PROGRAM MAIN
VAR CONSTANT
	INSTANCE_NAME: STRING := 'MAIN Program';
	IGNORE_DEFINITION: BOOL := TRUE;
	IGNORE_STOP: BOOL := TRUE;
END_VAR
VAR
	// define services
	m_buttonManager: ButtonManager;
	m_errorManager: ErrorManager;
	m_services: ServiceContainer(ADR(m_errorManager));
	
	// instantiate machine behavior model
	m_container: xPPU_Container(
		m_services.PtrStateTracker, 
		m_services.PtrProcessManager, 
		ADR(m_errorManager));
	
	// INTERLOCKS - must always be False
	// (EProcessVariables.LSC_RampEndWPCount >= 3) AND ((EProcessVariables.LSC_RampStartWPCount >= 3) OR ((EProcessVariables.LSC_RampMiddleWPCount >= 3) OR (EProcessVariables.SSC_RampWPCount >= 3)))
	m_compExpr1: ComparisonExpression(EProcessVariables.LSC_RampEndWPCount, EComparisonType.greater_eq, EDataType.numeric, FALSE, 3, '', TRUE);
	m_compExpr3: ComparisonExpression(EProcessVariables.LSC_RampStartWPCount, EComparisonType.greater_eq, EDataType.numeric, FALSE, 3, '', TRUE);
	m_compExpr5: ComparisonExpression(EProcessVariables.LSC_RampMiddleWPCount, EComparisonType.greater_eq, EDataType.numeric, FALSE, 3, '', TRUE);
	m_compExpr7: ComparisonExpression(EProcessVariables.SSC_RampWPCount, EComparisonType.greater_eq, EDataType.numeric, FALSE, 3, '', TRUE);
	m_boolExpr8: BoolExpression(m_compExpr5, EBoolOperation.or_op, m_compExpr7);
	m_boolExpr9: BoolExpression(m_compExpr3, EBoolOperation.or_op, m_boolExpr8);
	m_allRampsFull: BoolExpression(m_compExpr1, EBoolOperation.and_op, m_boolExpr9);
	
	// INTERLOCKS - must always be True
	// ...
	
	// MANUAL STRATEGY
	m_startAuto: BOOL;
	m_startManual: BOOL;
	m_stopManual: BOOL;
	m_strategyState: EOperationResult;
	
	// other
	i: UINT;
	m_statesEnum: EProcessVariables;
	m_emptyParams: ParameterSet;
	m_didFinishPrimitives: BOOL;
	m_appInitialized: BOOL;
	m_xPPU: xPPU_Automatic;
	m_customSeqStatus: EOperationResult;
	m_steps: ARRAY [0..2] OF STRING;
	m_appObservation: ARRAY[EProcessVariables.operating_mode..EProcessVariables.operating_mode] OF SValue;
END_VAR

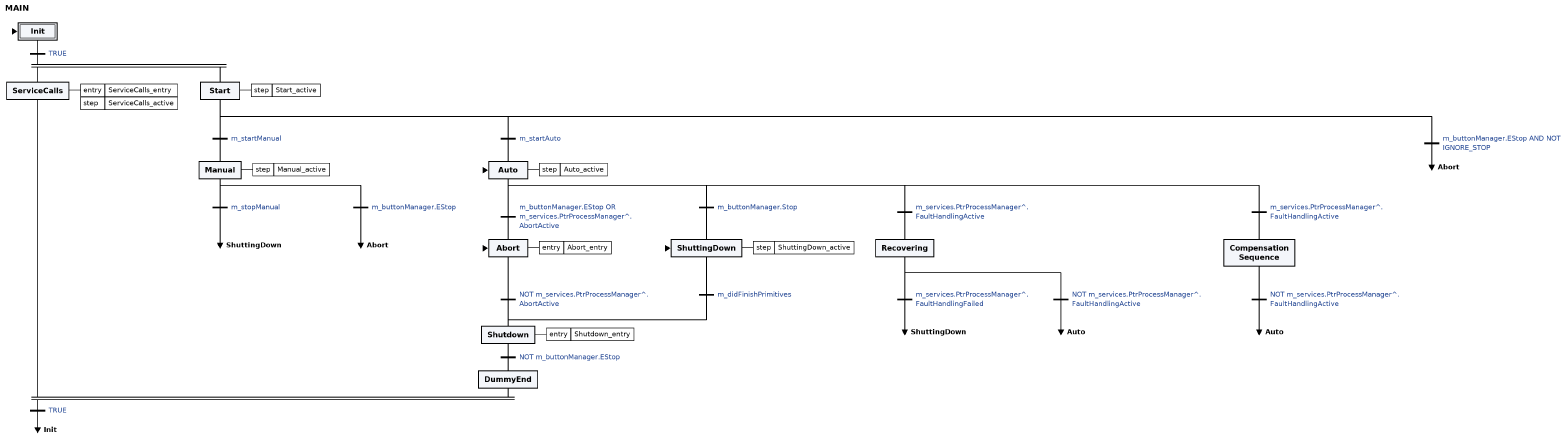
INITIAL_STEP Init:
END_STEP
TRANSITION FROM Init TO (ServiceCalls, Start)
    := TRUE;
END_TRANSITION
STEP ServiceCalls:
    ServiceCalls_entry(P1);  // entry action
    ServiceCalls_active(N);  // step action
END_STEP
STEP Start:
    Start_active(N);  // step action
END_STEP
TRANSITION FROM Start TO Manual
    := m_startManual;
END_TRANSITION
STEP Manual:
    Manual_active(N);  // step action
END_STEP
TRANSITION FROM Manual TO ShuttingDown
    := m_stopManual;
END_TRANSITION
TRANSITION FROM Manual TO Abort
    := m_buttonManager.EStop;
END_TRANSITION
TRANSITION FROM Start TO Auto
    := m_startAuto;
END_TRANSITION
STEP Auto:
    Auto_active(N);  // step action
END_STEP
TRANSITION FROM Auto TO Abort
    := m_buttonManager.EStop OR m_services.PtrProcessManager^.AbortActive;
END_TRANSITION
STEP Abort:
    Abort_entry(P1);  // entry action
END_STEP
TRANSITION FROM Abort TO Shutdown
    := NOT m_services.PtrProcessManager^.AbortActive;
END_TRANSITION
TRANSITION FROM Auto TO ShuttingDown
    := m_buttonManager.Stop;
END_TRANSITION
STEP ShuttingDown:
    ShuttingDown_active(N);  // step action
END_STEP
TRANSITION FROM ShuttingDown TO Shutdown
    := m_didFinishPrimitives;
END_TRANSITION
TRANSITION FROM Auto TO Recovering
    := m_services.PtrProcessManager^.FaultHandlingActive;
END_TRANSITION
STEP Recovering:
END_STEP
TRANSITION FROM Recovering TO ShuttingDown
    := m_services.PtrProcessManager^.FaultHandlingFailed;
END_TRANSITION
TRANSITION FROM Recovering TO Auto
    := NOT m_services.PtrProcessManager^.FaultHandlingActive;
END_TRANSITION
TRANSITION FROM Auto TO CompensationSequence
    := m_services.PtrProcessManager^.FaultHandlingActive;
END_TRANSITION
STEP CompensationSequence:
END_STEP
TRANSITION FROM CompensationSequence TO Auto
    := NOT m_services.PtrProcessManager^.FaultHandlingActive;
END_TRANSITION
STEP Shutdown:
    Shutdown_entry(P1);  // entry action
END_STEP
TRANSITION FROM Shutdown TO DummyEnd
    := NOT m_buttonManager.EStop;
END_TRANSITION
TRANSITION FROM Start TO Abort
    := m_buttonManager.EStop AND NOT IGNORE_STOP;
END_TRANSITION
STEP DummyEnd:
END_STEP
TRANSITION FROM (ServiceCalls, DummyEnd) TO Init
    := TRUE;
END_TRANSITION

ACTION Abort_entry:
m_services.PtrProcessManager^.RequestAbort();
END_ACTION

ACTION Auto_active:
m_xPPU(
	i_ptrErrorManager := m_services.PtrErrorManager,
	i_ptrProcessManager := m_services.PtrProcessManager,
	i_ptrStateTracker := m_services.PtrStateTracker);
END_ACTION

ACTION Manual_active:


m_strategyState := m_services.PtrProcessManager^.ExecuteCustomStrategy();
m_stopManual := m_buttonManager.Stop 
	OR NOT m_services.PtrProcessManager^.CustomStrategyReady 
	OR m_strategyState = EOperationResult.success;
END_ACTION

ACTION ServiceCalls_active:
// process state observation
m_appObservation[EProcessVariables.operating_mode].DataType := EDataType.string_t;
m_appObservation[EProcessVariables.operating_mode].Value.String_t := SFCCurrentStep;

// cylic service updates
IF m_services.PtrStateTracker <>0 THEN
m_services.PtrStateTracker^.CyclicUpdateStatus(IGNORE_DEFINITION,m_appObservation);
m_services.PtrProcessManager^.CyclicManageBehavior();
END_IF
END_ACTION

ACTION ServiceCalls_entry:
IF NOT m_appInitialized THEN
	FC_InitAlarmTexts();
	
	// init process variable names
	FOR i := ResiConst.ARR_MIN TO ResiConst.STATE_ARR_MAX DO
		m_statesEnum := i;
		m_services.PtrStateTracker^.SetProcessVariableName(i, TO_STRING(m_statesEnum));
	END_FOR
	
	// add interlocks
	m_services.PtrStateTracker^.AddInterlock(m_allRampsFull, FALSE);
	
	m_appInitialized := TRUE;
	m_errorManager.AddMessage(EAlarms.initialized, TRUE, ESeverity.info, 'MAIN');
END_IF
END_ACTION

ACTION Shutdown_entry:
m_errorManager.AddMessage(
	i_alarmId := EAlarms.stopped,
	i_active := TRUE,
	i_severity := ESeverity.info,
	i_instanceName := INSTANCE_NAME);

m_services.PtrStateTracker^.ResetDefinitions();
END_ACTION

ACTION ShuttingDown_active:
m_didFinishPrimitives := m_services.PtrProcessManager^.FinishPrimitives(i_abortRecoveries := TRUE);
END_ACTION

ACTION Start_active:
m_startManual := m_buttonManager.Mode = EOperatingModes.manual AND m_services.PtrProcessManager^.CustomStrategyReady AND m_buttonManager.Start;
m_startAuto := m_buttonManager.Mode = EOperatingModes.automatic AND m_buttonManager.Start;
END_ACTION

END_PROGRAM

(* stored: Version 1.1.0.1
   POU MAIN: Id {a58bb666-43ab-46d1-86a0-bca8bb16f09d}, SpecialFunc None
   Action Abort_entry: Id {99ab6845-5539-4711-8874-815ac3457b5b}
   Action Auto_active: Id {04ce01cc-9c38-475b-8a5a-1fc20fe7563e}
   Action Manual_active: Id {2d822a92-05f0-432c-a5a6-99bb4d17c0ba}
   Action ServiceCalls_active: Id {6606d316-b039-41b0-bf6b-5c561aa539c7}
   Action ServiceCalls_entry: Id {24c536b4-2fb2-44ef-8d75-892e48d5ec1d}
   Action Shutdown_entry: Id {056f07e9-48aa-4c4b-bb7b-3ccbd0dcc4b7}
   Action ShuttingDown_active: Id {b1b16c20-54da-4d9f-88a1-e95076766694}
   Action Start_active: Id {edc2770b-bafe-4378-a54c-e488f6b79a86} *)
